FUNCTION_BLOCK COLLAB_FOREST (* Peroidic event generator *)
  (* Standard: 61499-1 Annex A; Description: Copyright (c) 2017 fortiss GmbH This program and the accompanying materials are made available under the terms of the Eclipse Public License 2.0 which is available at https://www.eclipse.org/legal/epl-2.0/ SPDX-License-Identifier: EPL-2.0 *)
  (* Version 1.0, 2017-09-21, Alois Zoitl, fortiss GmbH, initial API and implementation and/or initial documentation *)
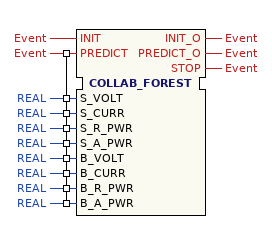
  EVENT_INPUT
    INIT;
    PREDICT WITH S_VOLT, S_CURR, S_R_PWR, S_A_PWR, B_VOLT, B_CURR, B_R_PWR, B_A_PWR;
  END_EVENT
  EVENT_OUTPUT
    INIT_O;
    PREDICT_O;
    STOP;
  END_EVENT
  VAR_INPUT
    S_VOLT : REAL;
    S_CURR : REAL;
    S_R_PWR : REAL;
    S_A_PWR : REAL;
    B_VOLT : REAL;
    B_CURR : REAL;
    B_R_PWR : REAL;
    B_A_PWR : REAL;
  END_VAR
END_FUNCTION_BLOCK
